{attribute 'qualified_only'}
{attribute 'strict'}
{attribute 'to_string'}
TYPE nTableBottlePlaceState :
(
	Empty := 0,
	BeforeWeighing := 1,
	Processing := 2,
	AfterWeighing := 3,
	NOK :=4,
	Drawer := 5,
	Tare := 6
);
END_TYPE

(* stored: Version 1.1.0.1, ProductVersion 3.1.4024.15
   DUT nTableBottlePlaceState: Id {e76810a4-c641-4fe2-9772-be01d895fc18} *)
